(* IEC 61131-3 sources: eCockpitGit/test_project/src/%F%02 System/%F%03 LoadSaveManager/%POU%FB_LoadSave/%F%Save/%F%Structure/%PRO%maxSize, 1 file *)

(* ---- %GETSET%Get.st ---- *)
//This gets the amount of bytes in the buffer
// | 1         | NSN      | 22-06-20 | Creation
VAR
END_VAR

(*%!%__DELIMITER__%!%*)
maxSize		:=		writer.maxSize;
